(* IEC 61131-3 sources: Industry-PLC-LLM/data/PLCBEAD_repo/PLCBEAD_PLCEmbed-main/PLC-BEAD/Source/GEB/DAY_OF_WEEK, 1 file *)

(* ---- DAY_OF_WEEK.ST ---- *)
FUNCTION DAY_OF_WEEK:INT
  VAR_INPUT
    IDATE :	UDINT;
  END_VAR

  DAY_OF_WEEK := UDINT_TO_INT((IDATE / UDINT#86400 + UDINT#3) MOD UDINT#7) + INT#01;
END_FUNCTION

PROGRAM program0
  VAR
    LocalVar0 : UDINT;
	LocalOUT  : INT;
  END_VAR
  	LocalOUT := DAY_OF_WEEK(LocalVar0);
END_PROGRAM
